(* PLC project Unnamed, Unknown Unnamed 1 *)
(* stored: creationDateTime 2024-08-24T11:36:06, modificationDateTime 2024-08-28T12:29:01 *)

PROGRAM Water_Tank
  VAR
    low_level_sensor : BOOL;  (* Input that indicates if the water level is below the minimum level. *)
    pump : BOOL;  (* Output that controls if the water pump if on or off. *)
    high_level_sensor : BOOL;  (* Input that indicates if the water level is above the maximum level. *)
    SR0 : SR;
  END_VAR

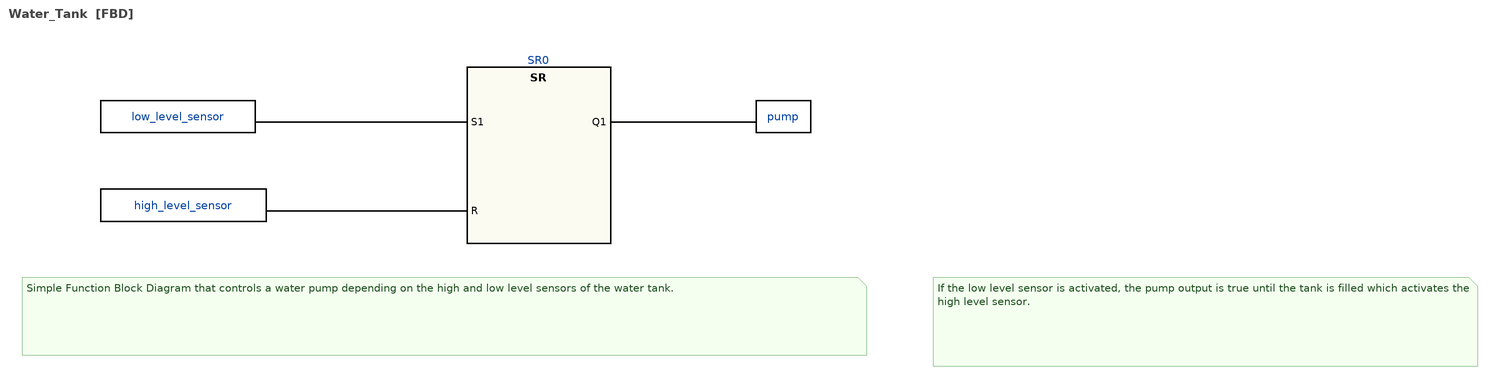
(* FBD diagram, written out as Structured Text *)
SR0(S1 := low_level_sensor, R := high_level_sensor);
pump := SR0.Q1;
(* Simple Function Block Diagram that controls a water pump depending on the high and low level sensors of the water tank. *)
(* If the low level sensor is activated, the pump output is true until the tank is filled which activates the high level sensor. *)
END_PROGRAM

CONFIGURATION Config0
  RESOURCE Res0 ON PLC
    TASK task0(INTERVAL := T#20ms, PRIORITY := 0);
    PROGRAM instance0 WITH task0 : Water_Tank;
  END_RESOURCE
END_CONFIGURATION
